(* CoDeSys 2.3 export: FESTOAR.EXP *)
(* Libraries: 3S_CanDrv.lib 10.6.10 10:53:10, 3S_CANOpenManager.lib 21.11.11 09:12:46, 3S_CANOpenMaster.lib 18.2.11 10:56:50, ANALYZATION.LIB 5.10.99 10:05:06, IECSFC.LIB 13.4.06 15:51:28, KAAD.lib 10.6.10 10:53:06, KDiagFunctions.lib 10.6.10 10:53:06, KMSG.lib 10.6.10 10:53:06, KSWO.lib 10.6.10 10:53:06, KSys.lib 10.6.10 10:53:20, KTypes.lib 10.6.10 10:53:06, McUtils.lib 24.5.12 15:38:58, PlcService.lib 10.6.10 10:53:20, RcInterface.lib 29.6.12 12:58:48, RcIntern.lib 24.5.12 15:38:58, RcSignalProcessing.lib 24.5.12 15:38:58, RcTracking.lib 24.5.12 15:38:58, STANDARD.LIB 4.10.05 12:14:46, SYSLIBCALLBACK.LIB 30.11.11 08:05:58, SysLibFile.lib 10.6.10 10:53:00, SysLibFileAsync.lib 21.11.11 09:12:46, SysLibIecTasks.lib 10.6.10 10:53:02, SysLibRtc.lib 10.6.10 10:53:02, SysLibSockets.lib 21.11.11 09:12:46, SysLibSocketsAsync.lib 21.11.11 09:12:46, SYSLIBTIME.LIB 10.6.10 10:53:02, SYSTASKINFO.LIB 10.6.10 10:53:02, ThreadSafeString.lib 14.5.12 16:17:26, Util.lib 18.5.10 15:14:28 *)

(* PLC configuration (modules and I/O channels)
Festo CMXR-C2 [Root] node -1, in %IB0 out %QB0 {param 1 = 1}
  Communication [Net] node 0, in %IB0 out %QB0 {param 1 = 0}
  ExtModules [IO] node 1, in %IB0 out %QB0 {param 1 = KBUS:0; param 2 = IX* STAT}
    AT %IX0.0 [ERR] bus error
    CECX-D-8E8A-NP-2 [DM272a] node 0, in %IB4 out %QB0 {param 1 = [0]; param 2 = 1; param 3 = none; param 4 = none; param 5 = none; param 6 = none; param 7 = none; param 8 = none; param 9 = none; param 10 = none; param 11 = none; param 12 = none; param 13 = none; param 14 = DM272A; param 15 = IX* DI +0; param 16 = .IX* DI +1; param 17 = .IX* DI +2; param 18 = .IX* DI +3; param 19 = .IX* DI +4; param 20 = .IX* DI +5; param 21 = .IX* DI +6; param 22 = .IX* DI +7; param 23 = QX* DO +0; param 24 = .QX* DO +1; param 25 = .QX* DO +2; param 26 = .QX* DO +3; param 27 = .QX* DO +4; param 28 = .QX* DO +5; param 29 = .QX* DO +6; param 30 = .QX* DO +7; param 31 = IX* STAT; param 32 = IX* DI.STAT +0; param 33 = .IX* DI.STAT +1; param 34 = .IX* DI.STAT +2; param 35 = .IX* DI.STAT +3; param 36 = .IX* DI.STAT +4; param 37 = .IX* DI.STAT +5; param 38 = .IX* DI.STAT +6; param 39 = .IX* DI.STAT +7; param 40 = IX* DO.STAT +0; param 41 = .IX* DO.STAT +1; param 42 = .IX* DO.STAT +2; param 43 = .IX* DO.STAT +3; param 44 = .IX* DO.STAT +4; param 45 = .IX* DO.STAT +5; param 46 = .IX* DO.STAT +6; param 47 = .IX* DO.STAT +7}
      dinEmStop AT %IX4.0 [DI]
      dinEnabling AT %IX4.1 [DI]
      dinAutoSelect AT %IX4.2 [DI]
      dinManSelect AT %IX4.3 [DI]
      DIO88_0_In_4 AT %IX4.4 [DI]
      DIO88_0_In_5 AT %IX4.5 [DI]
      DIO88_0_In_6 AT %IX4.6 [DI]
      DIO88_0_In_7 AT %IX4.7 [DI]
      doutError AT %QX0.0 [DO]
      DIO88_0_Out_1 AT %QX0.1 [DO]
      doutAutoSelected AT %QX0.2 [DO]
      doutManSelected AT %QX0.3 [DO]
      DIO88_0_Out_4 AT %QX0.4 [DO]
      DIO88_0_Out_5 AT %QX0.5 [DO]
      DIO88_0_Out_6 AT %QX0.6 [DO]
      DIO88_0_Out_7 AT %QX0.7 [DO]
      Module Status [DM272a_ERR] node 0, in %IB5 out %QB1
        DIO88_0_err AT %IX5.0 [ERB] Module error
        DI Status [ERR_DI8] node 0, in %IB6 out %QB1
          dinEmStop_err AT %IX6.0 [ERR] DI0 error
          dinEnabling_err AT %IX6.1 [ERR] DI1 error
          dinAutoSelect_err AT %IX6.2 [ERR] DI2 error
          dinManSelect_err AT %IX6.3 [ERR] DI3 error
          DIO88_0_In_4_err AT %IX6.4 [ERR] DI4 error
          DIO88_0_In_5_err AT %IX6.5 [ERR] DI5 error
          DIO88_0_In_6_err AT %IX6.6 [ERR] DI6 error
          DIO88_0_In_7_err AT %IX6.7 [ERR] DI7 error
        DO Status [ERR_DO8] node 1, in %IB7 out %QB1
          doutError_err AT %IX7.0 [ERR] DO0 error
          DIO88_0_Out_1_err AT %IX7.1 [ERR] DO1 error
          doutAutoSelected_err AT %IX7.2 [ERR] DO2 error
          doutManSelected_err AT %IX7.3 [ERR] DO3 error
          DIO88_0_Out_4_err AT %IX7.4 [ERR] DO4 error
          DIO88_0_Out_5_err AT %IX7.5 [ERR] DO5 error
          DIO88_0_Out_6_err AT %IX7.6 [ERR] DO6 error
          DIO88_0_Out_7_err AT %IX7.7 [ERR] DO7 error
  CAN Master X4 [FxCanMaster] node 2, in %IB8 out %QB4 {param 1 = UserTask}
*)

(* Task configuration *)
TASK MotionTask (PRIORITY := 1, INTERVAL := T#20ms);
  RC_INTERFACE();
END_TASK
TASK UserTask (PRIORITY := 10, INTERVAL := T#20ms);
  MAIN();
 RC_STANDALONE();
END_TASK
TASK UDPTCPExample (PRIORITY := 10, INTERVAL := T#200ms);
 TCPServer();
END_TASK

(* Global variable list: CanOpen implicit Variables *)
VAR_GLOBAL CONSTANT
	MAX_CTRLINDEX : INT := 0;
END_VAR
VAR_GLOBAL CONSTANT
	USE_CANOPEN_NODES : BOOL := FALSE;
	MAX_MASTERINDEX : INT := 0;
	MAX_NODEINDEX : INT := 0;
	MAX_SDOINDEX : INT := 0;
	MAX_PDOINDEX_RX : INT := 0;
	MAX_PDOINDEX_TX : INT := 0;
	MAX_MASTER_ODENTRY_IDX : INT := 0;
END_VAR
VAR_GLOBAL
	pCANopenMaster : ARRAY[0..MAX_MASTERINDEX] OF CanOpenMaster;
	pCanOpenNode : ARRAY[0..MAX_NODEINDEX] OF CanOpenNode;
	pCanOpenSDO : ARRAY[0..MAX_SDOINDEX] OF CanOpenSDO;
	pCanOpenPDO_Rx : ARRAY[0..MAX_PDOINDEX_RX] OF CanOpenPDO_Rx;
	pCanOpenPDO_Tx : ARRAY[0..MAX_PDOINDEX_TX] OF CanOpenPDO_Tx;
	 ODMEntries: ARRAY[0..MAX_MASTER_ODENTRY_IDX] OF CanOpenODEntry;
END_VAR

(* Global variable list: Global_Variables *)
VAR_GLOBAL
	TCPServerOnline: BOOL;
	SocketSrv: DINT;
	SocketCli: DINT;
	DataRcv: ARRAY[0..13] OF BYTE;
	RcvPacketCount: DINT;
	NbRcvBytes: DINT;
	DataSend: ARRAY[0..7] OF BYTE := 1,2,3,4,3,2,1,0;
	ReadDone: BOOL;
	ReadBusy: BOOL;
	Client : CLIENT_ACCEPT;
	RobotData: ROBOT_DATA;
END_VAR

(* Global variable list: RC_INTERFACE_INSTANCES *)
VAR_GLOBAL
(* Global Instances of RC_INTERFACE(PRG)                 *)
(* CDSA *)
	FBCDSAIfGetKeys          : CDSAIfGetKeys;
	FBCDSAIfSetProcessLed    : CDSAIfSetProcessLed;
(* Roboter Global *)
	FBRobotUpdateGlobal      : RcIfRobotUpdateGlobal;
	FBMsgRead                : RcIfMsgRead;
	FBMsgSet                 : RcIfMsgSet;
	FBMsgQuit                : RcIfMsgQuit;
	FBRegAxisPos             : RcIfRegAxisPos;
	FBRegCartPos             : RcIfRegCartPos;
(* Roboter Local *)
	FBRobotUpdateLocal       : RcIfRobotUpdateLocal;
	FBModeControl            : RcIfModeControl;
	FBRobotData              : RcIfRobotData;
	FBWriteAccess            : RcIfWriteAccess;
	FBJogControl             : RcIfJogControl;
	FBProgramControl         : RcIfProgramControl_V2;
	FBOverride               : RcIfOverride;
	FBSetRefSys              : RcIfSetRefSys;
	FBSetTool                : RcIfSetTool;
(*-------------------------------------------------------*)
END_VAR

(* Data type *)
TYPE CLIENT_ACCEPT :
STRUCT
	diSocket:DINT;
	stIPAddress:STRING(20);
END_STRUCT
END_TYPE

(* Data type *)
TYPE CLIENT_REPLY :
STRUCT
	diBytesReceived:DINT;
	stIPAddressTransmitter:STRING(20);
END_STRUCT
END_TYPE

(* Data type *)
TYPE ROBOT_DATA :
STRUCT
(* RcIfRobotData *)
	RobotName : STRING(80);
	RobotActive : BOOL;
	RobotReferenced : BOOL;
	RobotError : BOOL;
	RobotOverride : INT;
	RefSysName : STRING(80);
	RefSysNumber : DINT;
	Tool : TTool;
	ToolName : STRING(80);
	ToolNumber : DINT;
	AxisCountMain : DINT;
	AxisCountWrist : DINT;
	AxisCountAux : DINT;
	AxisSimulated : WORD;
	AxisReferenced : WORD;
	AxisLSN : WORD;
	AxisLSP : WORD;
	AxisPos : TAxisPos;
	CartPosWorld : TCARTPOS;
	CartPosRefSys : TCartPos;
	AxisDyn : TAxisDyn;
	PathDyn : TPathDyn;
	CartDyn : TCartDyn;
	Error : BOOL;
	ErrorId : TRcIfErrorID;
END_STRUCT
END_TYPE

(* POU RcInterface/RC_INTERFACE, FBD *)
PROGRAM RC_INTERFACE
VAR
(****************************************************************************************************************
     FESTO AG  Co., Esslingen                                                    								
     Copyright (c) 2009. All rights reserved.                       

  
 Program Name:   RC_INTERFACE 
 Description:    Programm for CoDeSys Controlinterface
 Composer:       FESTO
 Version:        00.01.02
 Last Change:    01.12.2011                                                                           
****************************************************************************************************************)
(* System Program please do not change *)

(****************************************************************************************************************
Change History

Date          Name                      Activity                                          Version                                                                  
                                                                                          
27.01.2010    bejk                      created                                           00.01.01
01.12.2011    bejk                      updated                                           00.01.02

****************************************************************************************************************)
END_VAR
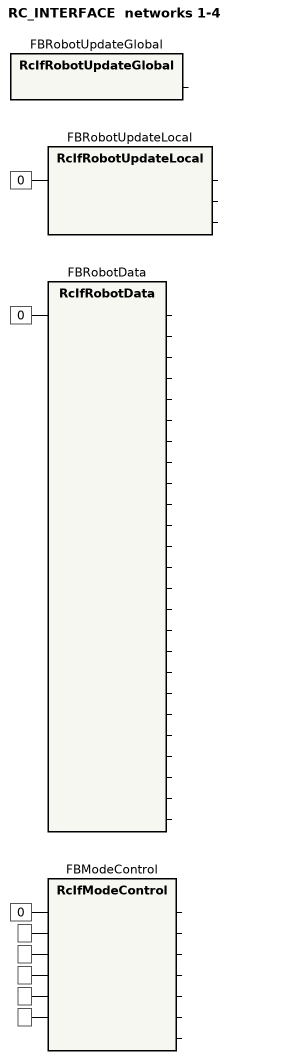
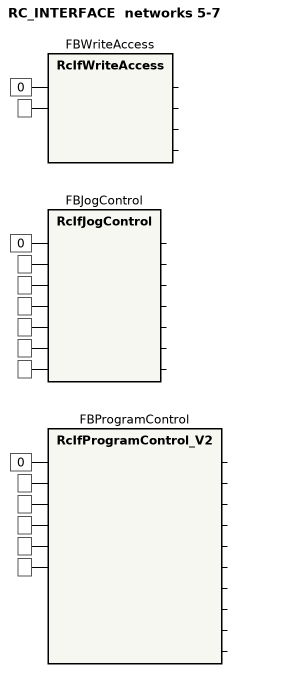
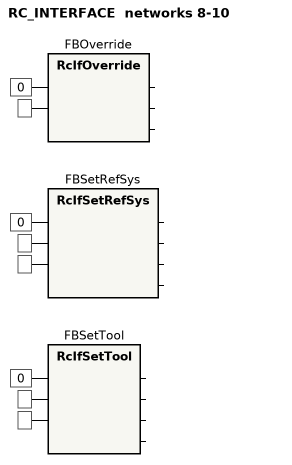
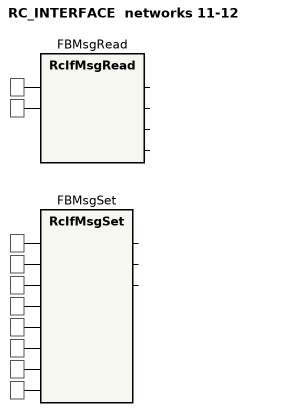
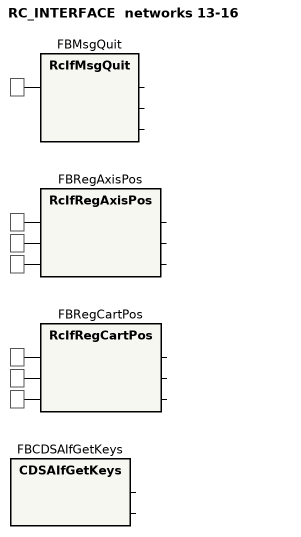
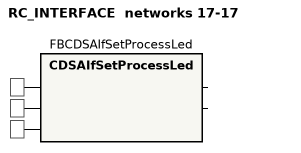
_FBD_ (* Function Block Diagram *)
NETWORK 1 (* RC_INTERFACE(PRG) *): (* Please do not change the system program, use the global instance variables to access the RC-Interface functions *)
	FBRobotUpdateGlobal:RcIfRobotUpdateGlobal()
NETWORK 2
	FBRobotUpdateLocal:RcIfRobotUpdateLocal(0)
NETWORK 3 (* Roboter local Function blocks *):
	FBRobotData:RcIfRobotData(0)
NETWORK 4
	FBModeControl:RcIfModeControl(0, , , , , )
NETWORK 5
	FBWriteAccess:RcIfWriteAccess(0, )
NETWORK 6
	FBJogControl:RcIfJogControl(0, , , , , , )
NETWORK 7
	FBProgramControl:RcIfProgramControl_V2(0, , , , , )
NETWORK 8
	FBOverride:RcIfOverride(0, )
NETWORK 9
	FBSetRefSys:RcIfSetRefSys(0, , )
NETWORK 10
	FBSetTool:RcIfSetTool(0, , )
NETWORK 11 (* Roboter global Function blocks *):
	FBMsgRead:RcIfMsgRead(, )
NETWORK 12
	FBMsgSet:RcIfMsgSet(, , , , , , , )
NETWORK 13
	FBMsgQuit:RcIfMsgQuit()
NETWORK 14
	FBRegAxisPos:RcIfRegAxisPos(, , )
NETWORK 15
	FBRegCartPos:RcIfRegCartPos(, , )
NETWORK 16 (* CDSA Functions *):
	FBCDSAIfGetKeys:CDSAIfGetKeys()
NETWORK 17
	FBCDSAIfSetProcessLed:CDSAIfSetProcessLed(, , )
_END_FBD_
(* the same logic as Structured Text *)
(* Network 1: see the listing above *)
(* Network 2 *)
FBRobotUpdateLocal(0);
(* Network 3: see the listing above *)
(* Network 4: see the listing above *)
(* Network 5: see the listing above *)
(* Network 6: see the listing above *)
(* Network 7: see the listing above *)
(* Network 8: see the listing above *)
(* Network 9: see the listing above *)
(* Network 10: see the listing above *)
(* Network 11: see the listing above *)
(* Network 12: see the listing above *)
(* Network 13: see the listing above *)
(* Network 14: see the listing above *)
(* Network 15: see the listing above *)
(* Network 16: see the listing above *)
(* Network 17: see the listing above *)
END_PROGRAM

(* POU MAIN, CFC *)
PROGRAM MAIN
VAR_IN_OUT
END_VAR
VAR
END_VAR
_CFC_ (* Continuous Function Chart, elements in execution order *)
(* ( * Add user Code here * ) *)
_END_CFC_
(* the same logic as Structured Text *)
(* ( * Add user Code here * ) *)
END_PROGRAM

(* POU RC_STANDALONE, CFC *)
PROGRAM RC_STANDALONE
(****************************************************************************************************************
     FESTO AG  Co., Esslingen                                                    								
     Copyright (c) 2009. All rights reserved.                       

  
 Program Name:   RC_STANDALONE 
 Description:    Example Programm how to use CMXR RC-Interface (variant standalone)
 Composer:       FESTO
 Version:        00.01.01
 Last Change:    31.08.2011                                                                           
****************************************************************************************************************)
(* Example Project how to use the RC-Interface *)

(****************************************************************************************************************
Change History

Date          Name                      Activity                                          Version                                                                  
                                                                                          
12.01.2010    bejk                      created                                           00.01.00
31.08.2011    bejk                      Bugfix FBRobotData.RobotError                     00.01.01
****************************************************************************************************************)
VAR
END_VAR
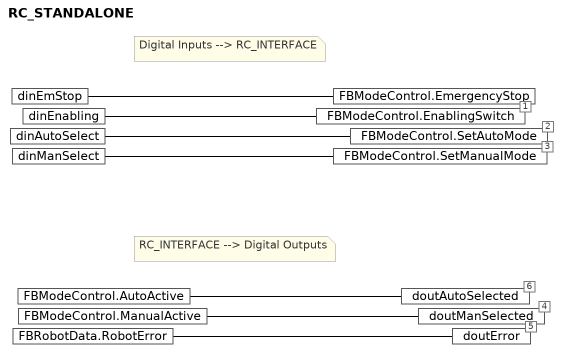
_CFC_ (* Continuous Function Chart, elements in execution order *)
(* Digital Inputs --> RC_INTERFACE *)
#0 FBModeControl.EmergencyStop <= dinEmStop
#1 FBModeControl.EnablingSwitch <= dinEnabling
#2 FBModeControl.SetAutoMode <= dinAutoSelect
#3 FBModeControl.SetManualMode <= dinManSelect
#4 doutManSelected <= FBModeControl.ManualActive
#5 doutError <= FBRobotData.RobotError
#6 doutAutoSelected <= FBModeControl.AutoActive
(* RC_INTERFACE --> Digital Outputs *)
_END_CFC_
(* the same logic as Structured Text *)
(* Digital Inputs --> RC_INTERFACE *)
FBModeControl.EmergencyStop := dinEmStop;
FBModeControl.EnablingSwitch := dinEnabling;
FBModeControl.SetAutoMode := dinAutoSelect;
FBModeControl.SetManualMode := dinManSelect;
doutManSelected := FBModeControl.ManualActive;
doutError := FBRobotData.RobotError;
doutAutoSelected := FBModeControl.AutoActive;
(* RC_INTERFACE --> Digital Outputs *)
END_PROGRAM

(* POU TCPServer, ST *)
PROGRAM TCPServer
VAR
	diSocket : DINT := -1;
	iPort : INT:=4508;
	Client : CLIENT_ACCEPT := (diSocket := -1);
	bySend : ARRAY[0..10] OF BYTE := 0,1,2,3,4,5,6,7,8,9,10;
	byData : STRING(10240); (* 10kB *)
	byRecv : ARRAY[0..14] OF BYTE;
	Reply : CLIENT_REPLY;
	bCloseClient: BOOL;
	bActive: BOOL:= TRUE;
END_VAR
byData := XMLPrinter();
IF bActive THEN
	IF diSocket = -1 THEN
		diSocket := TcpServerOpenSocket(iPort, 10, 1000);
	END_IF

	IF  Client.diSocket = -1 THEN
		Client := TcpServerWaitForConnect(diSocket, 4);
	END_IF

	IF  Client.diSocket <> -1 THEN
		TcpSendData(Client.diSocket, ADR(byData), SIZEOF(byData), 1);
		(*TcpReceiveData(Client.diSocket, ADR(byRecv), SIZEOF(byRecv), 5);*)
		bCloseClient := TRUE;
	END_IF

	IF bCloseClient THEN
		bCloseClient := FALSE;
		SysSockClose(diSocket:=Client.diSocket);
		Client.diSocket := -1;
	END_IF
END_IF
END_PROGRAM

(* POU FestoAR/XMLPrinter, ST *)
FUNCTION XMLPrinter : STRING
VAR_INPUT
END_VAR
VAR
	xml : STRING(10240); (* 10kB *)
END_VAR
xml := CONCAT(xml, '<root>');
xml := CONCAT(xml, '<RobotName>');
xml := CONCAT(xml, FBRobotData.RobotName);
xml := CONCAT(xml, '</RobotName>');
xml := CONCAT(xml, '<RobotActive>');
xml := CONCAT(xml, BOOL_TO_STRING(FBRobotData.RobotActive));
xml := CONCAT(xml, '</RobotActive>');
xml := CONCAT(xml, '<RobotReferenced>');
xml := CONCAT(xml, BOOL_TO_STRING(FBRobotData.RobotReferenced));
xml := CONCAT(xml, '</RobotReferenced>');
xml := CONCAT(xml, '<RobotError>');
xml := CONCAT(xml, BOOL_TO_STRING(FBRobotData.RobotError));
xml := CONCAT(xml, '</RobotError>');
xml := CONCAT(xml, '<RobotOverride>');
xml := CONCAT(xml, INT_TO_STRING(FBRobotData.RobotOverride));
xml := CONCAT(xml, '</RobotOverride>');
xml := CONCAT(xml, '<RefSysName>');
xml := CONCAT(xml, FBRobotData.RefSysName);
xml := CONCAT(xml, '</RefSysName>');
xml := CONCAT(xml, '<RefSysNumber>');
xml := CONCAT(xml, DINT_TO_STRING(FBRobotData.RefSysNumber));
xml := CONCAT(xml, '</RefSysNumber>');
xml := CONCAT(xml, '<Tool>');
xml := CONCAT(xml, '<x>');
xml := CONCAT(xml, REAL_TO_STRING(FBRobotData.Tool.x));
xml := CONCAT(xml, '</x>');
xml := CONCAT(xml, '<y>');
xml := CONCAT(xml, REAL_TO_STRING(FBRobotData.Tool.y));
xml := CONCAT(xml, '</y>');
xml := CONCAT(xml, '<z>');
xml := CONCAT(xml, REAL_TO_STRING(FBRobotData.Tool.z));
xml := CONCAT(xml, '</z>');
xml := CONCAT(xml, '<a>');
xml := CONCAT(xml, REAL_TO_STRING(FBRobotData.Tool.a));
xml := CONCAT(xml, '</a>');
xml := CONCAT(xml, '<b>');
xml := CONCAT(xml, REAL_TO_STRING(FBRobotData.Tool.b));
xml := CONCAT(xml, '</b>');
xml := CONCAT(xml, '<c>');
xml := CONCAT(xml, REAL_TO_STRING(FBRobotData.Tool.c));
xml := CONCAT(xml, '</c>');
xml := CONCAT(xml, '</Tool>');
xml := CONCAT(xml, '<ToolName>');
xml := CONCAT(xml, FBRobotData.ToolName);
xml := CONCAT(xml, '</ToolName>');
xml := CONCAT(xml, '<ToolNumber>');
xml := CONCAT(xml, DINT_TO_STRING(FBRobotData.ToolNumber));
xml := CONCAT(xml, '</ToolNumber>');
xml := CONCAT(xml, '<AxisCountMain>');
xml := CONCAT(xml, DINT_TO_STRING(FBRobotData.AxisCountMain));
xml := CONCAT(xml, '</AxisCountMain>');
xml := CONCAT(xml, '<AxisCountWrist>');
xml := CONCAT(xml, DINT_TO_STRING(FBRobotData.AxisCountWrist));
xml := CONCAT(xml, '</AxisCountWrist>');
xml := CONCAT(xml, '<AxisCountAux>');
xml := CONCAT(xml, DINT_TO_STRING(FBRobotData.AxisCountAux));
xml := CONCAT(xml, '</AxisCountAux>');
xml := CONCAT(xml, '<AxisSimulated>');
xml := CONCAT(xml, WORD_TO_STRING(FBRobotData.AxisSimulated));
xml := CONCAT(xml, '</AxisSimulated>');
xml := CONCAT(xml, '<AxisReferenced>');
xml := CONCAT(xml, WORD_TO_STRING(FBRobotData.AxisReferenced));
xml := CONCAT(xml, '</AxisReferenced>');
xml := CONCAT(xml, '<AxisLSN>');
xml := CONCAT(xml, WORD_TO_STRING(FBRobotData.AxisLSN));
xml := CONCAT(xml, '</AxisLSN>');
xml := CONCAT(xml, '<AxisLSP>');
xml := CONCAT(xml, WORD_TO_STRING(FBRobotData.AxisLSP));
xml := CONCAT(xml, '</AxisLSP>');
xml := CONCAT(xml, '<AxisPos>');
xml := CONCAT(xml, '<a1>');
xml := CONCAT(xml, REAL_TO_STRING(FBRobotData.AxisPos.a1));
xml := CONCAT(xml, '</a1>');
xml := CONCAT(xml, '<a2>');
xml := CONCAT(xml, REAL_TO_STRING(FBRobotData.AxisPos.a2));
xml := CONCAT(xml, '</a2>');
xml := CONCAT(xml, '<a3>');
xml := CONCAT(xml, REAL_TO_STRING(FBRobotData.AxisPos.a3));
xml := CONCAT(xml, '</a3>');
xml := CONCAT(xml, '<a4>');
xml := CONCAT(xml, REAL_TO_STRING(FBRobotData.AxisPos.a4));
xml := CONCAT(xml, '</a4>');
xml := CONCAT(xml, '<a5>');
xml := CONCAT(xml, REAL_TO_STRING(FBRobotData.AxisPos.a5));
xml := CONCAT(xml, '</a5>');
xml := CONCAT(xml, '<a6>');
xml := CONCAT(xml, REAL_TO_STRING(FBRobotData.AxisPos.a6));
xml := CONCAT(xml, '</a6>');
xml := CONCAT(xml, '<aux1>');
xml := CONCAT(xml, REAL_TO_STRING(FBRobotData.AxisPos.aux1));
xml := CONCAT(xml, '</aux1>');
xml := CONCAT(xml, '<aux2>');
xml := CONCAT(xml, REAL_TO_STRING(FBRobotData.AxisPos.aux2));
xml := CONCAT(xml, '</aux2>');
xml := CONCAT(xml, '<aux3>');
xml := CONCAT(xml, REAL_TO_STRING(FBRobotData.AxisPos.aux3));
xml := CONCAT(xml, '</aux3>');
xml := CONCAT(xml, '</AxisPos>');
xml := CONCAT(xml, '<CartPosWorld>');
xml := CONCAT(xml, '<x>');
xml := CONCAT(xml, REAL_TO_STRING(FBRobotData.CartPosWorld.x));
xml := CONCAT(xml, '</x>');
xml := CONCAT(xml, '<y>');
xml := CONCAT(xml, REAL_TO_STRING(FBRobotData.CartPosWorld.y));
xml := CONCAT(xml, '</y>');
xml := CONCAT(xml, '<z>');
xml := CONCAT(xml, REAL_TO_STRING(FBRobotData.CartPosWorld.z));
xml := CONCAT(xml, '</z>');
xml := CONCAT(xml, '<a>');
xml := CONCAT(xml, REAL_TO_STRING(FBRobotData.CartPosWorld.a));
xml := CONCAT(xml, '</a>');
xml := CONCAT(xml, '<b>');
xml := CONCAT(xml, REAL_TO_STRING(FBRobotData.CartPosWorld.b));
xml := CONCAT(xml, '</b>');
xml := CONCAT(xml, '<c>');
xml := CONCAT(xml, REAL_TO_STRING(FBRobotData.CartPosWorld.c));
xml := CONCAT(xml, '</c>');
xml := CONCAT(xml, '<aux1>');
xml := CONCAT(xml, REAL_TO_STRING(FBRobotData.CartPosWorld.aux1));
xml := CONCAT(xml, '</aux1>');
xml := CONCAT(xml, '<aux2>');
xml := CONCAT(xml, REAL_TO_STRING(FBRobotData.CartPosWorld.aux2));
xml := CONCAT(xml, '</aux2>');
xml := CONCAT(xml, '<aux3>');
xml := CONCAT(xml, REAL_TO_STRING(FBRobotData.CartPosWorld.aux3));
xml := CONCAT(xml, '</aux3>');
xml := CONCAT(xml, '</CartPosWorld>');
xml := CONCAT(xml, '<CartPosRefSys>');
xml := CONCAT(xml, '<x>');
xml := CONCAT(xml, REAL_TO_STRING(FBRobotData.CartPosRefSys.x));
xml := CONCAT(xml, '</x>');
xml := CONCAT(xml, '<y>');
xml := CONCAT(xml, REAL_TO_STRING(FBRobotData.CartPosRefSys.y));
xml := CONCAT(xml, '</y>');
xml := CONCAT(xml, '<z>');
xml := CONCAT(xml, REAL_TO_STRING(FBRobotData.CartPosRefSys.z));
xml := CONCAT(xml, '</z>');
xml := CONCAT(xml, '<a>');
xml := CONCAT(xml, REAL_TO_STRING(FBRobotData.CartPosRefSys.a));
xml := CONCAT(xml, '</a>');
xml := CONCAT(xml, '<b>');
xml := CONCAT(xml, REAL_TO_STRING(FBRobotData.CartPosRefSys.b));
xml := CONCAT(xml, '</b>');
xml := CONCAT(xml, '<c>');
xml := CONCAT(xml, REAL_TO_STRING(FBRobotData.CartPosRefSys.c));
xml := CONCAT(xml, '</c>');
xml := CONCAT(xml, '<aux1>');
xml := CONCAT(xml, REAL_TO_STRING(FBRobotData.CartPosRefSys.aux1));
xml := CONCAT(xml, '</aux1>');
xml := CONCAT(xml, '<aux2>');
xml := CONCAT(xml, REAL_TO_STRING(FBRobotData.CartPosRefSys.aux2));
xml := CONCAT(xml, '</aux2>');
xml := CONCAT(xml, '<aux3>');
xml := CONCAT(xml, REAL_TO_STRING(FBRobotData.CartPosRefSys.aux3));
xml := CONCAT(xml, '</aux3>');
xml := CONCAT(xml, '</CartPosRefSys>');
xml := CONCAT(xml, '<AxisDyn>');
xml := CONCAT(xml, '<a1>');
xml := CONCAT(xml, '<vel>');
xml := CONCAT(xml, REAL_TO_STRING(FBRobotData.AxisDyn.a1.vel));
xml := CONCAT(xml, '</vel>');
xml := CONCAT(xml, '<acc>');
xml := CONCAT(xml, REAL_TO_STRING(FBRobotData.AxisDyn.a1.acc));
xml := CONCAT(xml, '</acc>');
xml := CONCAT(xml, '<jerk>');
xml := CONCAT(xml, REAL_TO_STRING(FBRobotData.AxisDyn.a1.jerk));
xml := CONCAT(xml, '</jerk>');
xml := CONCAT(xml, '</a1>');
xml := CONCAT(xml, '<a2>');
xml := CONCAT(xml, '<vel>');
xml := CONCAT(xml, REAL_TO_STRING(FBRobotData.AxisDyn.a2.vel));
xml := CONCAT(xml, '</vel>');
xml := CONCAT(xml, '<acc>');
xml := CONCAT(xml, REAL_TO_STRING(FBRobotData.AxisDyn.a2.acc));
xml := CONCAT(xml, '</acc>');
xml := CONCAT(xml, '<jerk>');
xml := CONCAT(xml, REAL_TO_STRING(FBRobotData.AxisDyn.a2.jerk));
xml := CONCAT(xml, '</jerk>');
xml := CONCAT(xml, '</a2>');
xml := CONCAT(xml, '<a3>');
xml := CONCAT(xml, '<vel>');
xml := CONCAT(xml, REAL_TO_STRING(FBRobotData.AxisDyn.a3.vel));
xml := CONCAT(xml, '</vel>');
xml := CONCAT(xml, '<acc>');
xml := CONCAT(xml, REAL_TO_STRING(FBRobotData.AxisDyn.a3.acc));
xml := CONCAT(xml, '</acc>');
xml := CONCAT(xml, '<jerk>');
xml := CONCAT(xml, REAL_TO_STRING(FBRobotData.AxisDyn.a3.jerk));
xml := CONCAT(xml, '</jerk>');
xml := CONCAT(xml, '</a3>');
xml := CONCAT(xml, '<a4>');
xml := CONCAT(xml, '<vel>');
xml := CONCAT(xml, REAL_TO_STRING(FBRobotData.AxisDyn.a4.vel));
xml := CONCAT(xml, '</vel>');
xml := CONCAT(xml, '<acc>');
xml := CONCAT(xml, REAL_TO_STRING(FBRobotData.AxisDyn.a4.acc));
xml := CONCAT(xml, '</acc>');
xml := CONCAT(xml, '<jerk>');
xml := CONCAT(xml, REAL_TO_STRING(FBRobotData.AxisDyn.a4.jerk));
xml := CONCAT(xml, '</jerk>');
xml := CONCAT(xml, '</a4>');
xml := CONCAT(xml, '<a5>');
xml := CONCAT(xml, '<vel>');
xml := CONCAT(xml, REAL_TO_STRING(FBRobotData.AxisDyn.a5.vel));
xml := CONCAT(xml, '</vel>');
xml := CONCAT(xml, '<acc>');
xml := CONCAT(xml, REAL_TO_STRING(FBRobotData.AxisDyn.a5.acc));
xml := CONCAT(xml, '</acc>');
xml := CONCAT(xml, '<jerk>');
xml := CONCAT(xml, REAL_TO_STRING(FBRobotData.AxisDyn.a5.jerk));
xml := CONCAT(xml, '</jerk>');
xml := CONCAT(xml, '</a5>');
xml := CONCAT(xml, '<a6>');
xml := CONCAT(xml, '<vel>');
xml := CONCAT(xml, REAL_TO_STRING(FBRobotData.AxisDyn.a6.vel));
xml := CONCAT(xml, '</vel>');
xml := CONCAT(xml, '<acc>');
xml := CONCAT(xml, REAL_TO_STRING(FBRobotData.AxisDyn.a6.acc));
xml := CONCAT(xml, '</acc>');
xml := CONCAT(xml, '<jerk>');
xml := CONCAT(xml, REAL_TO_STRING(FBRobotData.AxisDyn.a6.jerk));
xml := CONCAT(xml, '</jerk>');
xml := CONCAT(xml, '</a6>');
xml := CONCAT(xml, '<aux1>');
xml := CONCAT(xml, '<vel>');
xml := CONCAT(xml, REAL_TO_STRING(FBRobotData.AxisDyn.aux1.vel));
xml := CONCAT(xml, '</vel>');
xml := CONCAT(xml, '<acc>');
xml := CONCAT(xml, REAL_TO_STRING(FBRobotData.AxisDyn.aux1.acc));
xml := CONCAT(xml, '</acc>');
xml := CONCAT(xml, '<jerk>');
xml := CONCAT(xml, REAL_TO_STRING(FBRobotData.AxisDyn.aux1.jerk));
xml := CONCAT(xml, '</jerk>');
xml := CONCAT(xml, '</aux1>');
xml := CONCAT(xml, '<aux2>');
xml := CONCAT(xml, '<vel>');
xml := CONCAT(xml, REAL_TO_STRING(FBRobotData.AxisDyn.aux2.vel));
xml := CONCAT(xml, '</vel>');
xml := CONCAT(xml, '<acc>');
xml := CONCAT(xml, REAL_TO_STRING(FBRobotData.AxisDyn.aux2.acc));
xml := CONCAT(xml, '</acc>');
xml := CONCAT(xml, '<jerk>');
xml := CONCAT(xml, REAL_TO_STRING(FBRobotData.AxisDyn.aux2.jerk));
xml := CONCAT(xml, '</jerk>');
xml := CONCAT(xml, '</aux2>');
xml := CONCAT(xml, '<aux3>');
xml := CONCAT(xml, '<vel>');
xml := CONCAT(xml, REAL_TO_STRING(FBRobotData.AxisDyn.aux3.vel));
xml := CONCAT(xml, '</vel>');
xml := CONCAT(xml, '<acc>');
xml := CONCAT(xml, REAL_TO_STRING(FBRobotData.AxisDyn.aux3.acc));
xml := CONCAT(xml, '</acc>');
xml := CONCAT(xml, '<jerk>');
xml := CONCAT(xml, REAL_TO_STRING(FBRobotData.AxisDyn.aux3.jerk));
xml := CONCAT(xml, '</jerk>');
xml := CONCAT(xml, '</aux3>');
xml := CONCAT(xml, '</AxisDyn>');
xml := CONCAT(xml, '<PathDyn>');
xml := CONCAT(xml, '<Path>');
xml := CONCAT(xml, '<vel>');
xml := CONCAT(xml, REAL_TO_STRING(FBRobotData.PathDyn.Path.vel));
xml := CONCAT(xml, '</vel>');
xml := CONCAT(xml, '<acc>');
xml := CONCAT(xml, REAL_TO_STRING(FBRobotData.PathDyn.Path.acc));
xml := CONCAT(xml, '</acc>');
xml := CONCAT(xml, '<jerk>');
xml := CONCAT(xml, REAL_TO_STRING(FBRobotData.PathDyn.Path.jerk));
xml := CONCAT(xml, '</jerk>');
xml := CONCAT(xml, '</Path>');
xml := CONCAT(xml, '<Ori>');
xml := CONCAT(xml, '<vel>');
xml := CONCAT(xml, REAL_TO_STRING(FBRobotData.PathDyn.Ori.vel));
xml := CONCAT(xml, '</vel>');
xml := CONCAT(xml, '<acc>');
xml := CONCAT(xml, REAL_TO_STRING(FBRobotData.PathDyn.Ori.acc));
xml := CONCAT(xml, '</acc>');
xml := CONCAT(xml, '<jerk>');
xml := CONCAT(xml, REAL_TO_STRING(FBRobotData.PathDyn.Ori.jerk));
xml := CONCAT(xml, '</jerk>');
xml := CONCAT(xml, '</Ori>');
xml := CONCAT(xml, '</PathDyn>');
xml := CONCAT(xml, '<CartDyn>');
xml := CONCAT(xml, '<x>');
xml := CONCAT(xml, '<vel>');
xml := CONCAT(xml, REAL_TO_STRING(FBRobotData.CartDyn.x.vel));
xml := CONCAT(xml, '</vel>');
xml := CONCAT(xml, '<acc>');
xml := CONCAT(xml, REAL_TO_STRING(FBRobotData.CartDyn.x.acc));
xml := CONCAT(xml, '</acc>');
xml := CONCAT(xml, '<jerk>');
xml := CONCAT(xml, REAL_TO_STRING(FBRobotData.CartDyn.x.jerk));
xml := CONCAT(xml, '</jerk>');
xml := CONCAT(xml, '</x>');
xml := CONCAT(xml, '<y>');
xml := CONCAT(xml, '<vel>');
xml := CONCAT(xml, REAL_TO_STRING(FBRobotData.CartDyn.y.vel));
xml := CONCAT(xml, '</vel>');
xml := CONCAT(xml, '<acc>');
xml := CONCAT(xml, REAL_TO_STRING(FBRobotData.CartDyn.y.acc));
xml := CONCAT(xml, '</acc>');
xml := CONCAT(xml, '<jerk>');
xml := CONCAT(xml, REAL_TO_STRING(FBRobotData.CartDyn.y.jerk));
xml := CONCAT(xml, '</jerk>');
xml := CONCAT(xml, '</y>');
xml := CONCAT(xml, '<z>');
xml := CONCAT(xml, '<vel>');
xml := CONCAT(xml, REAL_TO_STRING(FBRobotData.CartDyn.z.vel));
xml := CONCAT(xml, '</vel>');
xml := CONCAT(xml, '<acc>');
xml := CONCAT(xml, REAL_TO_STRING(FBRobotData.CartDyn.z.acc));
xml := CONCAT(xml, '</acc>');
xml := CONCAT(xml, '<jerk>');
xml := CONCAT(xml, REAL_TO_STRING(FBRobotData.CartDyn.z.jerk));
xml := CONCAT(xml, '</jerk>');
xml := CONCAT(xml, '</z>');
xml := CONCAT(xml, '<a>');
xml := CONCAT(xml, '<vel>');
xml := CONCAT(xml, REAL_TO_STRING(FBRobotData.CartDyn.a.vel));
xml := CONCAT(xml, '</vel>');
xml := CONCAT(xml, '<acc>');
xml := CONCAT(xml, REAL_TO_STRING(FBRobotData.CartDyn.a.acc));
xml := CONCAT(xml, '</acc>');
xml := CONCAT(xml, '<jerk>');
xml := CONCAT(xml, REAL_TO_STRING(FBRobotData.CartDyn.a.jerk));
xml := CONCAT(xml, '</jerk>');
xml := CONCAT(xml, '</a>');
xml := CONCAT(xml, '<b>');
xml := CONCAT(xml, '<vel>');
xml := CONCAT(xml, REAL_TO_STRING(FBRobotData.CartDyn.b.vel));
xml := CONCAT(xml, '</vel>');
xml := CONCAT(xml, '<acc>');
xml := CONCAT(xml, REAL_TO_STRING(FBRobotData.CartDyn.b.acc));
xml := CONCAT(xml, '</acc>');
xml := CONCAT(xml, '<jerk>');
xml := CONCAT(xml, REAL_TO_STRING(FBRobotData.CartDyn.b.jerk));
xml := CONCAT(xml, '</jerk>');
xml := CONCAT(xml, '</b>');
xml := CONCAT(xml, '<c>');
xml := CONCAT(xml, '<vel>');
xml := CONCAT(xml, REAL_TO_STRING(FBRobotData.CartDyn.c.vel));
xml := CONCAT(xml, '</vel>');
xml := CONCAT(xml, '<acc>');
xml := CONCAT(xml, REAL_TO_STRING(FBRobotData.CartDyn.c.acc));
xml := CONCAT(xml, '</acc>');
xml := CONCAT(xml, '<jerk>');
xml := CONCAT(xml, REAL_TO_STRING(FBRobotData.CartDyn.c.jerk));
xml := CONCAT(xml, '</jerk>');
xml := CONCAT(xml, '</c>');
xml := CONCAT(xml, '<aux1>');
xml := CONCAT(xml, '<vel>');
xml := CONCAT(xml, REAL_TO_STRING(FBRobotData.CartDyn.aux1.vel));
xml := CONCAT(xml, '</vel>');
xml := CONCAT(xml, '<acc>');
xml := CONCAT(xml, REAL_TO_STRING(FBRobotData.CartDyn.aux1.acc));
xml := CONCAT(xml, '</acc>');
xml := CONCAT(xml, '<jerk>');
xml := CONCAT(xml, REAL_TO_STRING(FBRobotData.CartDyn.aux1.jerk));
xml := CONCAT(xml, '</jerk>');
xml := CONCAT(xml, '</aux1>');
xml := CONCAT(xml, '<aux2>');
xml := CONCAT(xml, '<vel>');
xml := CONCAT(xml, REAL_TO_STRING(FBRobotData.CartDyn.aux2.vel));
xml := CONCAT(xml, '</vel>');
xml := CONCAT(xml, '<acc>');
xml := CONCAT(xml, REAL_TO_STRING(FBRobotData.CartDyn.aux2.acc));
xml := CONCAT(xml, '</acc>');
xml := CONCAT(xml, '<jerk>');
xml := CONCAT(xml, REAL_TO_STRING(FBRobotData.CartDyn.aux2.jerk));
xml := CONCAT(xml, '</jerk>');
xml := CONCAT(xml, '</aux2>');
xml := CONCAT(xml, '<aux3>');
xml := CONCAT(xml, '<vel>');
xml := CONCAT(xml, REAL_TO_STRING(FBRobotData.CartDyn.aux3.vel));
xml := CONCAT(xml, '</vel>');
xml := CONCAT(xml, '<acc>');
xml := CONCAT(xml, REAL_TO_STRING(FBRobotData.CartDyn.aux3.acc));
xml := CONCAT(xml, '</acc>');
xml := CONCAT(xml, '<jerk>');
xml := CONCAT(xml, REAL_TO_STRING(FBRobotData.CartDyn.aux3.jerk));
xml := CONCAT(xml, '</jerk>');
xml := CONCAT(xml, '</aux3>');
xml := CONCAT(xml, '</CartDyn>');
xml := CONCAT(xml, '<Error>');
xml := CONCAT(xml, BOOL_TO_STRING(FBRobotData.Error));
xml := CONCAT(xml, '</Error>');
xml := CONCAT(xml, '<ErrorId>');
xml := CONCAT(xml, DINT_TO_STRING(FBRobotData.ErrorId));
xml := CONCAT(xml, '</ErrorId>');
xml := CONCAT(xml, '</root>');

XMLPrinter := xml;
END_FUNCTION

(* POU Tcp specific/TcpServerOpenSocket, ST *)
FUNCTION TcpServerOpenSocket : DINT
(*	Open a TCP server socket.
	Return:	Main Socket Id
*)
VAR_INPUT
	iPort:INT;						(* Port number *)
	diMaxConnections:DINT;		(* Max possible client connections of the server *)
	diMaxDataSize:DINT;			(* Max size of data to transmitt; if size = 0 default values are used *)
END_VAR
VAR
	diSocket:DINT;
	bResult:BOOL;
	sa:SOCKADDRESS;
	bOptNoDelay:BOOL;
	lOptLinger:SOCKET_LINGER;
END_VAR
diSocket:=SysSockCreate(SOCKET_AF_INET, SOCKET_STREAM, SOCKET_IPPROTO_TCP);
IF diSocket <> SOCKET_INVALID THEN
(*
	IF diMaxDataSize <> 0 THEN
		SysSockSetOption(diSocket, SOCKET_SOL, SOCKET_SO_SNDBUF, ADR(diMaxDataSize), SIZEOF(diMaxDataSize));
		SysSockSetOption(diSocket, SOCKET_SOL, SOCKET_SO_RCVBUF, ADR(diMaxDataSize), SIZEOF(diMaxDataSize));
	END_IF
	lOptLinger.l_onoff:=0;
	lOptLinger.l_linger:=0;
	SysSockSetOption(diSocket,	SOCKET_SOL, SOCKET_SO_LINGER, ADR(lOptLinger), SIZEOF(lOptLinger));
	bOptNoDelay:=TRUE;
	SysSockSetOption(diSocket,	SOCKET_IPPROTO_TCP, SOCKET_TCP_NODELAY, ADR(bOptNoDelay), SIZEOF(bOptNoDelay));
*)

	sa.sin_family:=SOCKET_AF_INET;
	sa.sin_addr:=SOCKET_INADDR_ANY;
	sa.sin_port:=SysSockHtons(iPort);
	bResult:=SysSockBind(diSocket, ADR(sa), SIZEOF(sa));
	IF bResult = FALSE THEN
		diSocket:=SOCKET_INVALID;
	ELSE
		bResult:=SysSockListen(diSocket, diMaxConnections);
		IF bResult = FALSE THEN
			diSocket:=SOCKET_INVALID;
		END_IF
	END_IF
END_IF
TcpServerOpenSocket:=diSocket;
END_FUNCTION

(* POU Tcp specific/TcpServerWaitForConnect, ST *)
FUNCTION TcpServerWaitForConnect : CLIENT_ACCEPT
(*	Wait for a TCP client to connect.
	ATTENTION:  Function is blocking, until a client tries to connect!
	Return:	diSocket : Socket Id for connection session
				stIPAddress : IP-Address of connected client
*)
VAR_INPUT
	diServerSocket:DINT;
	diTimeout : DINT;	(* Timeout in seconds *)
END_VAR
VAR
	sa:SOCKADDRESS;
	ia:INADDR;
	diSize:DINT;
	fdRead: SOCKET_FD_SET;
	fdWrite:SOCKET_FD_SET;
	fdExcept:SOCKET_FD_SET;
	tvTimeout:SOCKET_TIMEVAL;
END_VAR
tvTimeout.tv_sec := diTimeout ;
tvTimeout.tv_usec := 0;
fdRead.fd_count := 1;
fdRead.fd_array[0] := diServerSocket;
IF (SysSockSelect(SOCKET_FD_SETSIZE, ADR(fdRead), 0, 0, ADR(tvTimeout)) > 0) THEN
	diSize:=SIZEOF(sa);
	TcpServerWaitForConnect.diSocket:=SysSockAccept(diServerSocket, ADR(sa), ADR(diSize));
	ia.S_addr:=UDINT_TO_DWORD(sa.sin_addr); (* Daniel: DINT_TO_DWORD -> UDINT_TO_DWORD *)
	SysSockInetNtoa(ia, TcpServerWaitForConnect.stIPAddress, SIZEOF(TcpServerWaitForConnect.stIPAddress));
ELSE
	TcpServerWaitForConnect.diSocket := -1;
END_IF
END_FUNCTION

(* POU Tcp specific/TcpSendData, ST *)
FUNCTION TcpSendData : DINT
(*	Send data via TCP socket.
	Return:	Number of bytes sent
*)
VAR_INPUT
	diSocket:DINT;		(* Socket Id *)
	pbyData:DWORD;		(* Address of data buffer *)
	diDataSize:DINT;		(* Size of data to send *)
	diTimeout : DINT;		(* Timeout in seconds *)
END_VAR
VAR
	fdWrite:SOCKET_FD_SET;
	tvTimeout:SOCKET_TIMEVAL;
END_VAR
tvTimeout.tv_sec := diTimeout ;
tvTimeout.tv_usec := 0;
fdWrite.fd_count := 1;
fdWrite.fd_array[0] := diSocket;
IF (SysSockSelect(SOCKET_FD_SETSIZE, 0, ADR(fdWrite), 0, ADR(tvTimeout)) > 0) THEN
	TcpSendData:=SysSockSend(diSocket, pbyData, diDataSize, 0);
END_IF
END_FUNCTION

(* POU RcInterface/RC_OUTPUT_UPDATE, ST *)
FUNCTION RC_OUTPUT_UPDATE : DWORD
VAR_INPUT
	dwEvent:DWORD;
	dwFilter:DWORD;
	dwOwner:DWORD;
END_VAR
IF NOT RcIfIosMapped THEN
	RcIfIosMapped := TRUE;

END_IF;
END_FUNCTION

(* POU Tcp specific/TcpReceiveData, ST *)
FUNCTION TcpReceiveData : DINT
(*	Receive data from a tcp socket.
	Return:	Number of bytes received
*)
VAR_INPUT
	diSocket:DINT;		(* Socket Id *)
	pbyData:DWORD;		(* Address of data buffer *)
	diDataSize:DINT;		(* Size of data to send *)
	diTImeout : DINT;		(* Timeout in seconds *)
END_VAR
VAR
	fdRead:SOCKET_FD_SET;
	tvTimeout:SOCKET_TIMEVAL;
END_VAR
tvTimeout.tv_sec := diTimeout ;
tvTimeout.tv_usec := 0;
fdRead.fd_count := 1;
fdRead.fd_array[0] := diSocket;
IF (SysSockSelect(SOCKET_FD_SETSIZE, ADR(fdRead), 0, 0, ADR(tvTimeout)) > 0) THEN
	TcpReceiveData:=SysSockRecv(diSocket, pbyData, diDataSize, 0);
END_IF
END_FUNCTION

(* Visualisation VISU_CDSA
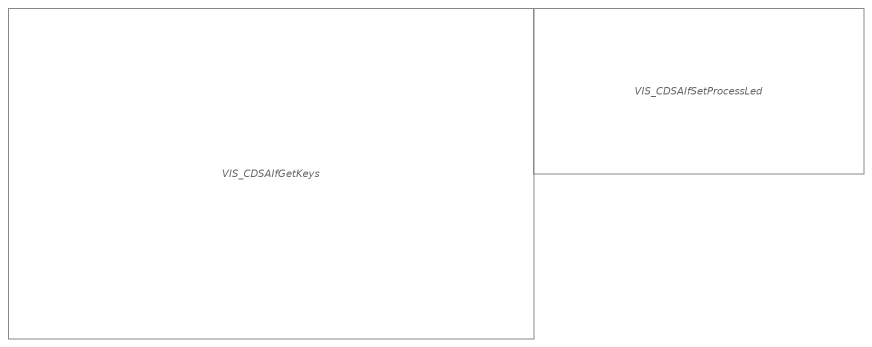
embedded screen at (0,0)-(526,331): VIS_CDSAIfGetKeys
embedded screen at (525,0)-(856,166): VIS_CDSAIfSetProcessLed
*)

(* Visualisation VISU_RegAccess
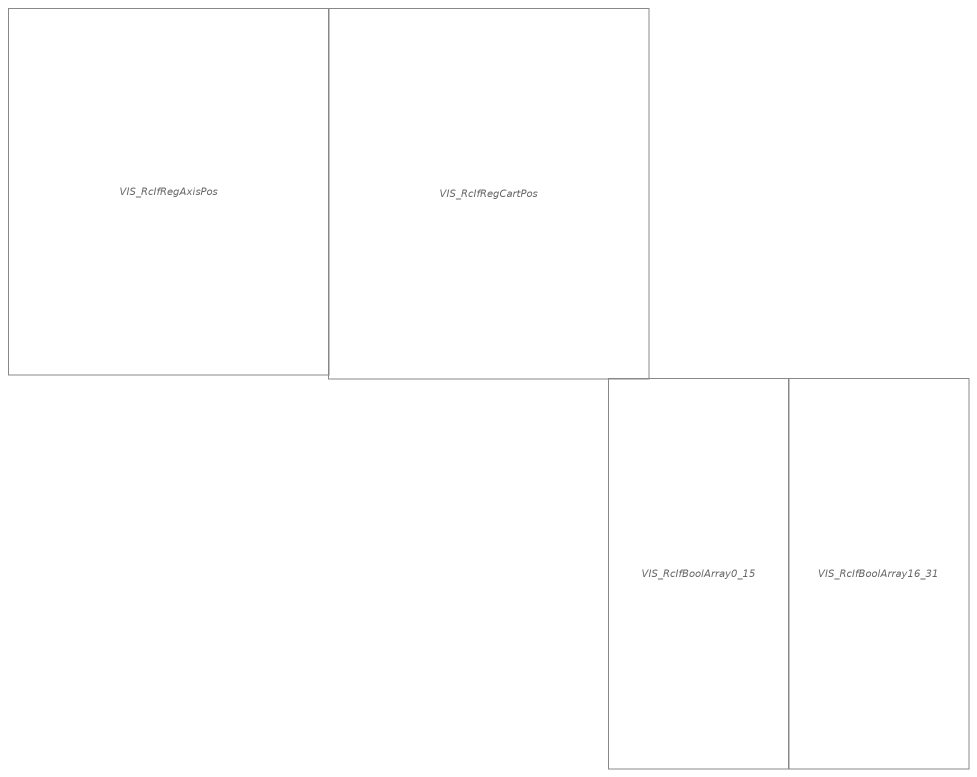
embedded screen at (320,0)-(641,371): VIS_RcIfRegCartPos
embedded screen at (600,370)-(781,761): VIS_RcIfBoolArray0_15
embedded screen at (780,370)-(961,761): VIS_RcIfBoolArray16_31
embedded screen at (0,0)-(321,367): VIS_RcIfRegAxisPos
*)

(* Visualisation VISU_RobotAxis
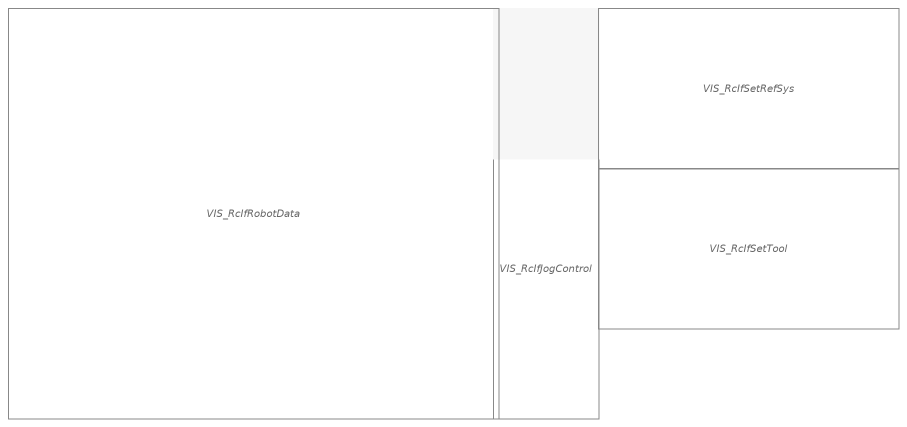
embedded screen at (485,110)-(591,411): VIS_RcIfJogControl
embedded screen at (0,0)-(491,411): VIS_RcIfRobotData
embedded screen at (590,0)-(891,161): VIS_RcIfSetRefSys
embedded screen at (590,160)-(891,321): VIS_RcIfSetTool
1 more shapes without text or variables
*)

(* Visualisation VISU_RobotControl
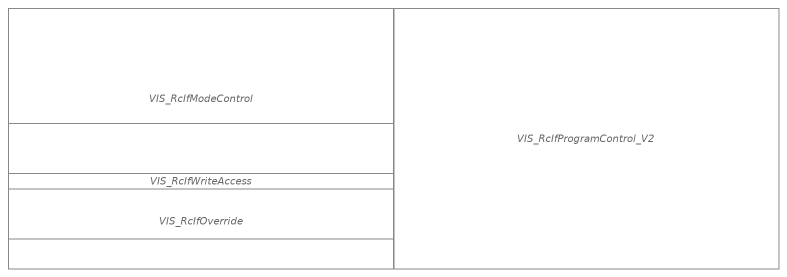
embedded screen at (0,165)-(386,261): VIS_RcIfOverride
embedded screen at (0,115)-(386,231): VIS_RcIfWriteAccess
embedded screen at (0,0)-(386,181): VIS_RcIfModeControl
embedded screen at (385,0)-(771,261): VIS_RcIfProgramControl_V2
*)

(* Visualisation VISU_RobotMessage
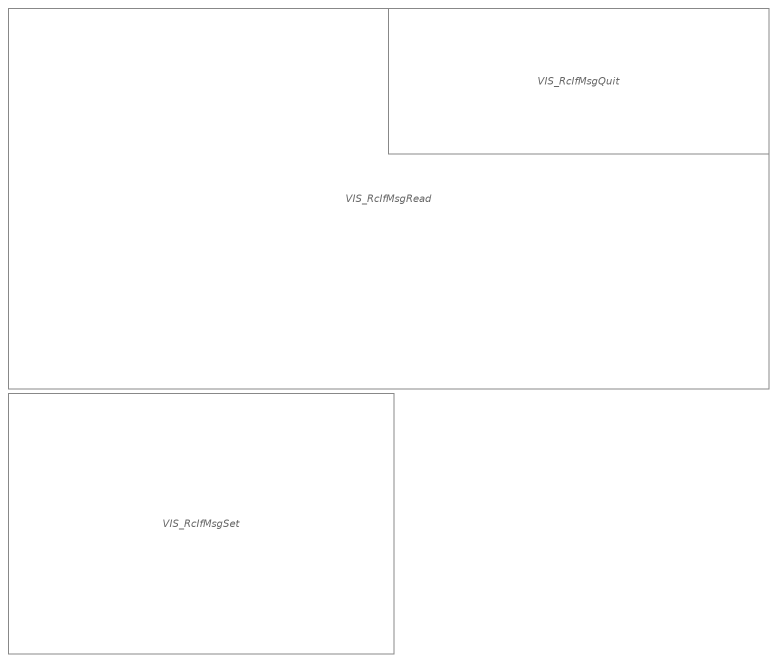
embedded screen at (0,0)-(761,381): VIS_RcIfMsgRead
embedded screen at (0,385)-(386,646): VIS_RcIfMsgSet
embedded screen at (380,0)-(761,146): VIS_RcIfMsgQuit
*)
